(* IEC 61131-3 sources: Word/plc-course/16-alarms-and-diagnostics/labs/solutions, 3 files *)

(* ---- 16-1-alarm-block.st ---- *)
(* Lab 16-1: FB_Alarm - one alarm with an on-delay, optional latching,
   edge-triggered acknowledge and reset, and the alarm states an HMI needs.
   Module 16 (Alarms, diagnostics and fault handling). REFERENCE SOLUTION - try the lab yourself first.

   Design: an alarm has two independent properties.
     Active  - is the alarm condition there (or, for a latching alarm, still latched)?
     Unacked - has the operator acknowledged the latest activation?
   The State output combines them, plus "has the condition gone?" for a
   latching alarm, into one value that an HMI can show directly. *)

TYPE
  E_AlarmState : (
    Normal,        (* not active, nothing to acknowledge *)
    ActiveUnack,   (* active, not yet acknowledged: flash + horn *)
    ActiveAcked,   (* active, acknowledged, condition still present: steady *)
    RtnUnack,      (* returned to normal before anyone acknowledged it *)
    LatchedRtn     (* latching alarm: acknowledged, condition gone, waiting for reset *)
  );
END_TYPE

FUNCTION_BLOCK FB_Alarm
  (* ------------------------------------------------------------------
     FB_Alarm - one annunciated alarm.

     Behaviour   Condition must last OnDelay before the alarm activates.
                 Each activation sets Active and Unacked and adds 1 to Count.
                 Ack (press) clears Unacked. Non-latching: Active follows
                 the confirmed condition. Latching: Active stays TRUE until
                 a Reset press while acknowledged and the condition is gone.
                 Reset never acknowledges and never affects a non-latching
                 alarm.
     Version     1.0  first release
     ------------------------------------------------------------------ *)
  VAR_INPUT
    Condition : BOOL;   (* raw alarm condition from the process logic *)
    OnDelay   : TIME;   (* Condition must last this long before the alarm activates *)
    Latching  : BOOL;   (* TRUE: stays active after the condition clears, until Reset *)
    Ack       : BOOL;   (* acknowledge command: acts on its rising edge *)
    Reset     : BOOL;   (* reset command for a latching alarm: acts on its rising edge *)
  END_VAR
  VAR_OUTPUT
    Active    : BOOL;   (* alarm is active: confirmed condition, or latched *)
    Unacked   : BOOL;   (* the latest activation has not been acknowledged *)
    State     : E_AlarmState;
    Count     : DINT;   (* activations since power-up, for alarm statistics *)
  END_VAR
  VAR
    DelayTimer : TON;
    AckEdge    : R_TRIG;
    ResetEdge  : R_TRIG;
    Confirmed  : BOOL;  (* Condition has lasted for OnDelay *)
  END_VAR

  (* 1. Confirm the condition. Any gap restarts the delay, so a fleeting
        condition shorter than OnDelay never reaches the operator. *)
  DelayTimer(IN := Condition, PT := OnDelay);
  Confirmed := DelayTimer.Q;

  AckEdge(CLK := Ack);
  ResetEdge(CLK := Reset);

  (* 2. Acknowledge BEFORE new activations are processed: a press can only
        acknowledge alarms that existed before it. Acting on the edge means
        a held or jammed button cannot acknowledge alarms that come later. *)
  IF AckEdge.Q THEN
    Unacked := FALSE;
  END_IF;

  (* 3. Return to normal. *)
  IF NOT Confirmed THEN
    IF NOT Latching THEN
      Active := FALSE;            (* Unacked is kept: "returned to normal, unacknowledged" *)
    ELSIF ResetEdge.Q AND NOT Unacked THEN
      Active := FALSE;            (* latched: only an acknowledged reset clears it *)
    END_IF;
  END_IF;

  (* 4. Activation: a confirmed condition on an alarm that is not active is
        a new occurrence, which the operator must acknowledge again. A
        latching alarm that is still latched is already active, so the
        condition coming back is not a new occurrence. *)
  IF Confirmed AND NOT Active THEN
    Active := TRUE;
    Unacked := TRUE;
    Count := Count + 1;
  END_IF;

  (* 5. One state value for the HMI. *)
  IF Active AND Unacked THEN
    State := ActiveUnack;
  ELSIF Active AND Confirmed THEN
    State := ActiveAcked;
  ELSIF Active THEN
    State := LatchedRtn;
  ELSIF Unacked THEN
    State := RtnUnack;
  ELSE
    State := Normal;
  END_IF;
END_FUNCTION_BLOCK

PROGRAM AlarmDemo
  VAR (* panel push-buttons and horn *)
    AckPB   AT %IX0.0 : BOOL;   (* Acknowledge push-button, NO *)
    ResetPB AT %IX0.1 : BOOL;   (* Reset push-button, NO *)
    Horn    AT %QX0.0 : BOOL;   (* Alarm horn *)
  END_VAR
  VAR (* alarm conditions: in a real program they come from process logic
         (for example FB_AnalogAlarm, Lab 14-2). Here the test writes them. *)
    TempHigh : BOOL;   (* TT-201 compressor bearing temperature high *)
    VibHigh  : BOOL;   (* VT-202 compressor vibration high-high *)
    DoorOpen : BOOL;   (* acoustic enclosure door open *)
  END_VAR
  VAR
    TempAlm : FB_Alarm;
    VibAlm  : FB_Alarm;
    DoorAlm : FB_Alarm;
  END_VAR

  (* The program is complete in the starter: only FB_Alarm is to be written. *)
  TempAlm(Condition := TempHigh, OnDelay := T#3s, Latching := FALSE, Ack := AckPB, Reset := ResetPB);
  VibAlm(Condition := VibHigh, OnDelay := T#1s, Latching := TRUE, Ack := AckPB, Reset := ResetPB);
  DoorAlm(Condition := DoorOpen, OnDelay := T#0s, Latching := FALSE, Ack := AckPB, Reset := ResetPB);

  (* The horn sounds while any alarm is unacknowledged. *)
  Horn := TempAlm.Unacked OR VibAlm.Unacked OR DoorAlm.Unacked;
END_PROGRAM

CONFIGURATION Config0
  RESOURCE Res0 ON PLC
    TASK MainTask(INTERVAL := T#10ms, PRIORITY := 0);
    PROGRAM Inst0 WITH MainTask : AlarmDemo;
  END_RESOURCE
END_CONFIGURATION

(* ---- 16-3-frozen-signal-heartbeat.st ---- *)
(* Lab 16-3: Frozen-signal and heartbeat diagnostics.
   Module 16 (Alarms, diagnostics and fault handling). REFERENCE SOLUTION - try the lab yourself first.

   Two small diagnostic blocks that catch faults a range check cannot see:
     FB_FrozenSignal  a transmitter value that stops moving while the
                      process is running (stuck sensor, transmitter left in
                      fixed-current mode, frozen communication value)
     FB_Heartbeat     a partner's heartbeat counter that stops changing
                      (partner stopped, or the link between us is down)
   The program also produces this PLC's own heartbeat for its partners. *)

FUNCTION_BLOCK FB_FrozenSignal
  (* ------------------------------------------------------------------
     FB_FrozenSignal - "has this value stopped moving?"

     Behaviour   While Enable is TRUE, Frozen goes TRUE when PV has stayed
                 within +/- Tolerance of a reference value for FreezeTime.
                 The reference is the PV at the last significant move (or
                 when Enable came on), NOT the previous scan's PV, so a
                 slow drift adds up and counts as movement. Any move of
                 more than Tolerance takes a new reference, restarts the
                 time and clears Frozen. Enable FALSE: no check, Frozen
                 FALSE. Frozen does not latch.
     Assumptions A live signal normally moves by more than Tolerance
                 within FreezeTime while Enable is TRUE (noise, pulsation,
                 normal process variation).
     Version     1.0  first release
     ------------------------------------------------------------------ *)
  VAR_INPUT
    PV         : REAL;   (* value to watch, engineering units *)
    Tolerance  : REAL;   (* a change larger than this counts as movement *)
    FreezeTime : TIME;   (* no movement for this long = frozen *)
    Enable     : BOOL;   (* TRUE while the process should make PV move *)
  END_VAR
  VAR_OUTPUT
    Frozen     : BOOL;   (* PV has not moved by more than Tolerance for FreezeTime *)
  END_VAR
  VAR
    RefValue   : REAL;   (* PV at the last significant move *)
    Moved      : BOOL;   (* PV moved more than Tolerance away from RefValue this scan *)
    StillTimer : TON;    (* time since the last significant move *)
  END_VAR

  IF NOT Enable THEN
    RefValue := PV;      (* keep the reference fresh while the check is off *)
    Moved := FALSE;
  ELSE
    Moved := ABS(PV - RefValue) > Tolerance;
    IF Moved THEN
      RefValue := PV;    (* new reference: measure the next move from here *)
    END_IF;
  END_IF;

  (* IN goes FALSE for one scan on every move, which restarts the timer.
     While disabled the timer is held at zero, so the full FreezeTime
     starts again when Enable comes back. *)
  StillTimer(IN := Enable AND NOT Moved, PT := FreezeTime);
  Frozen := StillTimer.Q;
END_FUNCTION_BLOCK

FUNCTION_BLOCK FB_Heartbeat
  (* ------------------------------------------------------------------
     FB_Heartbeat - supervise a heartbeat counter from a partner.

     Behaviour   Any change of Counter from one scan to the next is a
                 heartbeat: up, down, wrap-around or a reset to 0 after the
                 partner restarts. CommFault = no change for Timeout
                 (counted from power-up until the first change). CommOK =
                 a change has been seen within the last Timeout; it is
                 FALSE after power-up until the first change, because the
                 first value read is not proof that the partner is alive.
     Version     1.0  first release
     ------------------------------------------------------------------ *)
  VAR_INPUT
    Counter   : INT;     (* heartbeat counter received from the partner *)
    Timeout   : TIME;    (* no change for this long = partner or link lost *)
  END_VAR
  VAR_OUTPUT
    CommOK    : BOOL;    (* partner proven alive within the last Timeout *)
    CommFault : BOOL;    (* no change for Timeout: raise an alarm *)
  END_VAR
  VAR
    Started     : BOOL;  (* FALSE until the first call *)
    LastCounter : INT;   (* Counter on the previous scan *)
    Changed     : BOOL;  (* Counter changed since the previous scan *)
    SeenChange  : BOOL;  (* at least one change since power-up *)
    SilentTimer : TON;   (* time since the last change *)
  END_VAR

  IF NOT Started THEN
    LastCounter := Counter;   (* first scan: there is no earlier value to compare with *)
    Started := TRUE;
  END_IF;

  (* "Different", not "greater": a counter that wraps from 32767 to -32768,
     or restarts from 0, is still alive. *)
  Changed := Counter <> LastCounter;
  LastCounter := Counter;
  IF Changed THEN
    SeenChange := TRUE;
  END_IF;

  SilentTimer(IN := NOT Changed, PT := Timeout);
  CommFault := SilentTimer.Q;
  CommOK := SeenChange AND NOT SilentTimer.Q;
END_FUNCTION_BLOCK

PROGRAM PumpDiagnostics
  VAR (* I/O *)
    PumpRunFb AT %IX0.0 : BOOL;   (* P-301 contactor auxiliary contact: TRUE = running *)
    FrozenAlm AT %QX0.0 : BOOL;   (* a transmitter looks frozen *)
    CommAlm   AT %QX0.1 : BOOL;   (* a heartbeat has been lost *)
  END_VAR
  VAR (* values from the analog input blocks (Lab 14-1) and the communication
         driver (Module 17). Here the test writes them directly. *)
    PT301        : REAL;   (* P-301 discharge pressure, bar *)
    FT302        : REAL;   (* P-301 discharge flow, m3/h *)
    PartnerHB    : INT;    (* heartbeat counter from PLC-2: it adds 1 every second *)
    ScadaHB      : INT;    (* watchdog counter the SCADA server writes every few seconds *)
    HeartbeatOut : INT;    (* this PLC's own heartbeat, read by PLC-2 and SCADA *)
  END_VAR
  VAR
    PT301Chk   : FB_FrozenSignal;
    FT302Chk   : FB_FrozenSignal;
    PartnerMon : FB_Heartbeat;
    ScadaMon   : FB_Heartbeat;
    BeatTimer  : TON;
  END_VAR

  (* A running pump's discharge pressure and flow always move a little
     (pulsation, turbulence). When the pump is stopped they may be dead
     steady, so the check only runs while the pump runs. *)
  PT301Chk(PV := PT301, Tolerance := 0.05, FreezeTime := T#10s, Enable := PumpRunFb);
  FT302Chk(PV := FT302, Tolerance := 0.5, FreezeTime := T#20s, Enable := PumpRunFb);

  (* PLC-2 counts once a second: 3 s allows two missed updates.
     SCADA writes more slowly and less regularly: 10 s. *)
  PartnerMon(Counter := PartnerHB, Timeout := T#3s);
  ScadaMon(Counter := ScadaHB, Timeout := T#10s);

  FrozenAlm := PT301Chk.Frozen OR FT302Chk.Frozen;
  CommAlm := PartnerMon.CommFault OR ScadaMon.CommFault;

  (* Our own heartbeat: add 1 every second. The explicit wrap keeps the
     counter out of integer overflow, which some platforms report as a
     fault. For the receiver any change is a heartbeat, so the jump from
     32767 back to 0 is fine. *)
  BeatTimer(IN := NOT BeatTimer.Q, PT := T#1s);
  IF BeatTimer.Q THEN
    IF HeartbeatOut >= 32767 THEN
      HeartbeatOut := 0;
    ELSE
      HeartbeatOut := HeartbeatOut + 1;
    END_IF;
  END_IF;
END_PROGRAM

CONFIGURATION Config0
  RESOURCE Res0 ON PLC
    TASK MainTask(INTERVAL := T#10ms, PRIORITY := 0);
    PROGRAM Inst0 WITH MainTask : PumpDiagnostics;
  END_RESOURCE
END_CONFIGURATION

(* ---- 16-2-first-out-annunciator.st ---- *)
(* Lab 16-2: First-out annunciator for the eight shutdown inputs of a gas
   compressor, with horn, acknowledge, reset, lamp test and a run permissive.
   Module 16 (Alarms, diagnostics and fault handling). REFERENCE SOLUTION - try the lab yourself first.

   TRAINING EXERCISE ONLY: on a real compressor the shutdown function itself
   belongs in a properly designed (often safety-rated) trip system. This lab
   is about annunciation: showing the operator what tripped, and what
   tripped FIRST.

   Design: the eight inputs are copied into an array once per scan, and
   every rule is then a FOR loop over the channels. The order of the steps
   inside the scan is part of the design:
     1. acknowledge   (a press only acknowledges what was there before it)
     2. reset         (only acknowledged channels whose input is healthy)
     3. armed?        (worked out ONCE, before any new trip is latched)
     4. latch new trips, and mark them first-out if the panel was armed
     5. lamps, horn and run permissive *)

PROGRAM FirstOutPanel
  VAR (* trip inputs: NC contacts, TRUE = healthy, FALSE = tripped or wire broken *)
    Trip1_NC   AT %IX0.0 : BOOL;  (* PSLL-401 suction pressure low-low *)
    Trip2_NC   AT %IX0.1 : BOOL;  (* PSHH-402 discharge pressure high-high *)
    Trip3_NC   AT %IX0.2 : BOOL;  (* TSHH-403 discharge temperature high-high *)
    Trip4_NC   AT %IX0.3 : BOOL;  (* PSLL-404 lube oil pressure low-low *)
    Trip5_NC   AT %IX0.4 : BOOL;  (* VSHH-405 vibration high-high *)
    Trip6_NC   AT %IX0.5 : BOOL;  (* LSHH-406 suction scrubber level high-high *)
    Trip7_NC   AT %IX0.6 : BOOL;  (* HS-407 local shutdown push-button (monitoring contact) *)
    Trip8_NC   AT %IX0.7 : BOOL;  (* XA-408 main motor protection relay trip *)
    AckPB      AT %IX1.0 : BOOL;  (* Acknowledge (silence) push-button, NO *)
    ResetPB    AT %IX1.1 : BOOL;  (* Reset push-button, NO *)
    LampTestPB AT %IX1.2 : BOOL;  (* Lamp test push-button, NO *)
    Lamp1      AT %QX0.0 : BOOL;  (* annunciator window lamps, one per channel *)
    Lamp2      AT %QX0.1 : BOOL;
    Lamp3      AT %QX0.2 : BOOL;
    Lamp4      AT %QX0.3 : BOOL;
    Lamp5      AT %QX0.4 : BOOL;
    Lamp6      AT %QX0.5 : BOOL;
    Lamp7      AT %QX0.6 : BOOL;
    Lamp8      AT %QX0.7 : BOOL;
    Horn       AT %QX1.0 : BOOL;  (* audible alarm *)
    RunPermit  AT %QX1.1 : BOOL;  (* TRUE = compressor may be started (no channel latched) *)
  END_VAR
  VAR (* status for the HMI, one element per channel *)
    Latched  : ARRAY[1..8] OF BOOL;  (* channel has tripped and has not been reset *)
    Unacked  : ARRAY[1..8] OF BOOL;  (* channel trip not yet acknowledged *)
    FirstOut : ARRAY[1..8] OF BOOL;  (* channel was (one of) the first to trip *)
  END_VAR
  VAR
    Healthy    : ARRAY[1..8] OF BOOL;  (* copy of the eight NC inputs *)
    LampState  : ARRAY[1..8] OF BOOL;  (* lamp outputs before mapping to %QX *)
    AckEdge    : R_TRIG;
    ResetEdge  : R_TRIG;
    FlashTimer : TON;
    FlashOn    : BOOL;   (* toggles about every 0.5 s *)
    Armed      : BOOL;   (* no channel latched: the next trip is a first-out *)
    AnyLatched : BOOL;
    AnyUnacked : BOOL;
    I          : INT;
  END_VAR

  (* Input mapping: one place where the hardware meets the logic. *)
  Healthy[1] := Trip1_NC;
  Healthy[2] := Trip2_NC;
  Healthy[3] := Trip3_NC;
  Healthy[4] := Trip4_NC;
  Healthy[5] := Trip5_NC;
  Healthy[6] := Trip6_NC;
  Healthy[7] := Trip7_NC;
  Healthy[8] := Trip8_NC;

  AckEdge(CLK := AckPB);
  ResetEdge(CLK := ResetPB);

  (* 1. Acknowledge all channels on the PRESS of the button. A held button
        does not acknowledge trips that arrive later. *)
  IF AckEdge.Q THEN
    FOR I := 1 TO 8 DO
      Unacked[I] := FALSE;
    END_FOR;
  END_IF;

  (* 2. Reset clears only channels that are acknowledged AND healthy. A
        channel whose input is still tripped stays latched, with its
        first-out flag, so the evidence is not lost. *)
  IF ResetEdge.Q THEN
    FOR I := 1 TO 8 DO
      IF Healthy[I] AND NOT Unacked[I] THEN
        Latched[I] := FALSE;
        FirstOut[I] := FALSE;
      END_IF;
    END_FOR;
  END_IF;

  (* 3. Armed = nothing latched at this point of the scan. Decide it ONCE,
        before latching anything, so that every channel tripping in this
        scan is treated the same: within one scan the PLC cannot tell
        which came first, so they are all first-outs. *)
  Armed := TRUE;
  FOR I := 1 TO 8 DO
    IF Latched[I] THEN
      Armed := FALSE;
    END_IF;
  END_FOR;

  (* 4. Latch new trips. A channel that is already latched ignores its
        input until it has been reset. *)
  FOR I := 1 TO 8 DO
    IF (NOT Healthy[I]) AND (NOT Latched[I]) THEN
      Latched[I] := TRUE;
      Unacked[I] := TRUE;
      FirstOut[I] := Armed;
    END_IF;
  END_FOR;

  (* 5. Flasher: FlashOn toggles each time the timer runs out (about every
        0.5 s; the timer restarts on the scan after it finishes). *)
  FlashTimer(IN := NOT FlashTimer.Q, PT := T#500ms);
  IF FlashTimer.Q THEN
    FlashOn := NOT FlashOn;
  END_IF;

  (* 6. Lamps: flashing = needs attention (unacknowledged) or is the first
        cause; steady = acknowledged subsequent trip; off = not latched.
        The lamp test lights every lamp and changes nothing else. *)
  AnyLatched := FALSE;
  AnyUnacked := FALSE;
  FOR I := 1 TO 8 DO
    AnyLatched := AnyLatched OR Latched[I];
    AnyUnacked := AnyUnacked OR Unacked[I];
    IF LampTestPB THEN
      LampState[I] := TRUE;
    ELSIF Latched[I] AND (Unacked[I] OR FirstOut[I]) THEN
      LampState[I] := FlashOn;
    ELSE
      LampState[I] := Latched[I];
    END_IF;
  END_FOR;

  Horn := AnyUnacked;
  (* The permissive only ALLOWS a start. Reset never starts the compressor:
     that needs a separate, deliberate start command elsewhere. *)
  RunPermit := NOT AnyLatched;

  (* Output mapping *)
  Lamp1 := LampState[1];
  Lamp2 := LampState[2];
  Lamp3 := LampState[3];
  Lamp4 := LampState[4];
  Lamp5 := LampState[5];
  Lamp6 := LampState[6];
  Lamp7 := LampState[7];
  Lamp8 := LampState[8];
END_PROGRAM

CONFIGURATION Config0
  RESOURCE Res0 ON PLC
    TASK MainTask(INTERVAL := T#10ms, PRIORITY := 0);
    PROGRAM Inst0 WITH MainTask : FirstOutPanel;
  END_RESOURCE
END_CONFIGURATION
